FUNCTION_BLOCK SuspendedToHaltedUnifiedProgramTransition EXTENDS SuspendedToHaltedProgramTransition
VAR
	{attribute 'OPC.UA.DA' := '0'}
	_ClassName : STRING := __POUNAME();
END_VAR

{attribute 'monitoring' := 'call'}
PROPERTY ClassName : STRING
GET
ClassName := _ClassName;
END_GET
END_PROPERTY

END_FUNCTION_BLOCK

(* stored: Version 1.1.0.1
   POU SuspendedToHaltedUnifiedProgramTransition: Id {7df02ca3-2909-46c0-963e-8fd0302bf218}, SpecialFunc None
   Property ClassName: Id {75be853b-212d-4f49-985d-7fce2eda429e}
   Get Get: Id {3c5df878-3730-4ad0-8521-d9180c3e3412} *)
